TYPE ST_OutputStationHSUpcomingConfigurationOP11600 :
STRUCT
	{attribute 'OPC.UA.DA.Description' := 'Number of tools configured for the operation (0-200)'}
	ToolCapacityUsed			: UINT;

	{attribute 'OPC.UA.DA.Description' := 'IDs of upcoming tools'}
	{attribute 'OPC.UA.DA.StructuredType' := '1'}
	Tool 						: ARRAY [1..200] OF ToolX;

	{attribute 'OPC.UA.DA.Description' := 'Upcoming number of material configured for the operation (0-200)'}
	MaterialCapacityUsed		: UINT; 

	{attribute 'OPC.UA.DA.Description' := 'IDs OF upcoming material'}
	Material					: ARRAY [1..200] OF STRING(30);

END_STRUCT
END_TYPE

(* stored: Version 1.1.0.1, ProductVersion 3.1.4024.2
   DUT ST_OutputStationHSUpcomingConfigurationOP11600: Id {c6541e98-a2c2-45c4-a2aa-802bc9161dd8} *)
